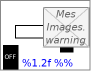
VISUALIZATION VISU_SOURCE_EFFET_JOULE  // 91x71
VAR_IN_OUT
	m_Input_SOURCE : BLOCK_SOURCE_JOULE;
END_VAR
    Polygon (30,49)
    Rectangle (15,57 65x12), "%1.2f %%", text variable: m_Input_SOURCE.STATE_POWER
    Polyline (69,38)
    Polyline (20,37)
    Rectangle (15,25 48x13)
    Polyline (65,41), colour toggle: m_Input_SOURCE.EJ.STATE_ON
    Rectangle (4,45 13x22), "ON", invisible if: NOT m_Input_SOURCE.STATE_EJ_ON
    Rectangle (4,46 13x22), "OFF", invisible if: m_Input_SOURCE.STATE_EJ_ON
    Rectangle (3,45 15x24), invisible if: NOT m_Input_SOURCE.EJ.AUTOR_ON_IHM AND NOT m_Input_SOURCE.EJ.AUTOR_OFF_IHM, input disabled if: (NOT m_Input_SOURCE.EJ.AUTOR_ON_IHM AND NOT m_Input_SOURCE.EJ.AUTOR_OFF_IHM) OR NOT PRG_User.ACTU_USER.MAINTENANCE
        tap m_Input_SOURCE.EJ.M_On
    Polygon (45,28), invisible if: NOT ( m_Input_SOURCE.EJ.STATE_On AND (m_Input_SOURCE.STATE_power > 0) )
    Rectangle (60,47 13x5), colour toggle: m_Input_SOURCE.WATER
    Image (43,7 46x40), invisible if: NOT m_Input_SOURCE.STATE_NOK, image: MesImages.warning
END_VISUALIZATION

(* stored: Version 1.1.0.1, ProductVersion 3.1.4024.10
   Visu VISU_SOURCE_EFFET_JOULE: Id {0ed4d9da-c075-49c8-a432-5d63cc5601a8} *)
